PROGRAM MAIN
VAR
END_VAR

END_PROGRAM

(* stored: Version 1.1.0.1
   POU MAIN: Id {1f160e3d-12a5-48fd-9295-7f020309da4e} *)
